// TwinCAT 3 PLC project MAS418_PLC
// ProgramVersion: 3.1.4024.0
// libraries:
//   Tc2_Standard, * (Beckhoff Automation GmbH)
//   Tc2_System, * (Beckhoff Automation GmbH)
//   Tc3_Module, * (Beckhoff Automation GmbH)
//   VisuDialogs, * (System)
// project tree:
//   / GlobalTextList.TcGTLO, PlcTask.TcTTO, Visualization Manager.TcVMO (not stored)
//   POUs/ MAIN.TcPOU
//   VISUs/ HMI.TcVIS

CONFIGURATION MAS418_PLC
    RESOURCE PLC ON TwinCAT3
        TASK PlcTask(INTERVAL := T#10ms, PRIORITY := 20);
        PROGRAM MAIN WITH PlcTask : MAIN;
    END_RESOURCE
END_CONFIGURATION

// ---- POUs/MAIN.TcPOU
PROGRAM MAIN
VAR
	bEnable : BOOL;
	bStart : BOOL;
	
	nINT : INT := -32768;
	nUINT : UINT := 65535;
	fREAL : REAL := 255.255;
	sPowerStatus: STRING := 'Power Off'; 
	
END_VAR


bEnable := bStart;

END_PROGRAM

// ---- GlobalTextList.TcGTLO
TEXTLIST GlobalTextList
  859 = '%f'
  129 = '%i'
  88 = '%s'
  651 = 'BOOL'
  605 = 'DataTypeTesting'
  766 = 'GroupBox'
  13 = 'POWER ON'
END_TEXTLIST

// ---- VISUs/HMI.TcVIS
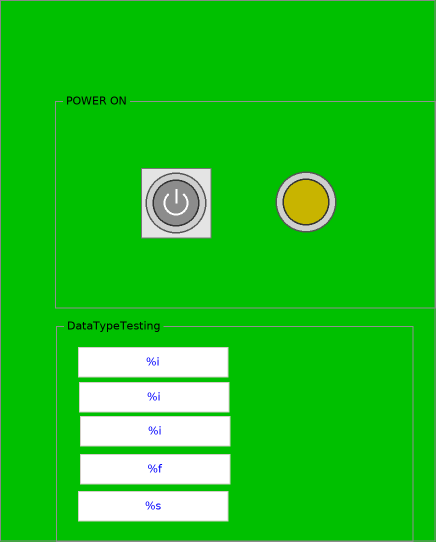
VISUALIZATION HMI  // 436x542
    GroupBox (55,93 381x215), "POWER ON"
        Lamp1 (216,74 70x70), variable: MAIN.bEnable, style: Lamp-Lamp1-Yellow
        PowerSwitch (86,75 70x70), variable: MAIN.bStart, behaviour: TOGGLE, style: Switch-PowerSwitch-Gray
    GroupBox (56,318 357x224), "DataTypeTesting"
        Textfield (22,29 150x30), "%i", text variable: MAIN.bEnable
        Textfield (23,64 150x30), "%i", text variable: MAIN.nINT
        Textfield (22,173 150x30), "%s", text variable: MAIN.sPowerStatus
            OnMouseDown: write the text variable via Default
        Textfield (24,136 150x30), "%f", text variable: MAIN.fREAL
            OnMouseDown: write the text variable via Default, min 0, max 1
        Textfield (24,98 150x30), "%i", text variable: MAIN.nUINT
END_VISUALIZATION
